Staubli VAL3: HOME.dtx

public TrajHome tTraj{}
  [home]
    num nIndexTool
    TrajJointItem tData
      [0]
        jointRx jJoint
        TrajectoryItem tSuper
          [0]
            num distance
            num moveType
            num nTime
            num nStop
            num nTcpAction
            string comment
            bool toStop
            mdesc nom_speed = {vel=50, tmax=500}
            InstrItem iInstr[3]
              [0]
                string sType
                string sData
              [1]
                string sType
                string sData
              [2]
                string sType
                string sData
            num nMoveId
    string sID = "home"
    num nZoneType
    num nZoneMove
    pointRx pO = {fatherId=world[0]}
    pointRx pX = {fatherId=world[0]}
    pointRx pY = {fatherId=world[0]}
    num nDimension
    pointRx pPointMove = {fatherId=tTraj["home"].fFrame[0]}
    frame fFrame = {fatherId=world[0]}
    string sProgram
    num nIndexFrame
